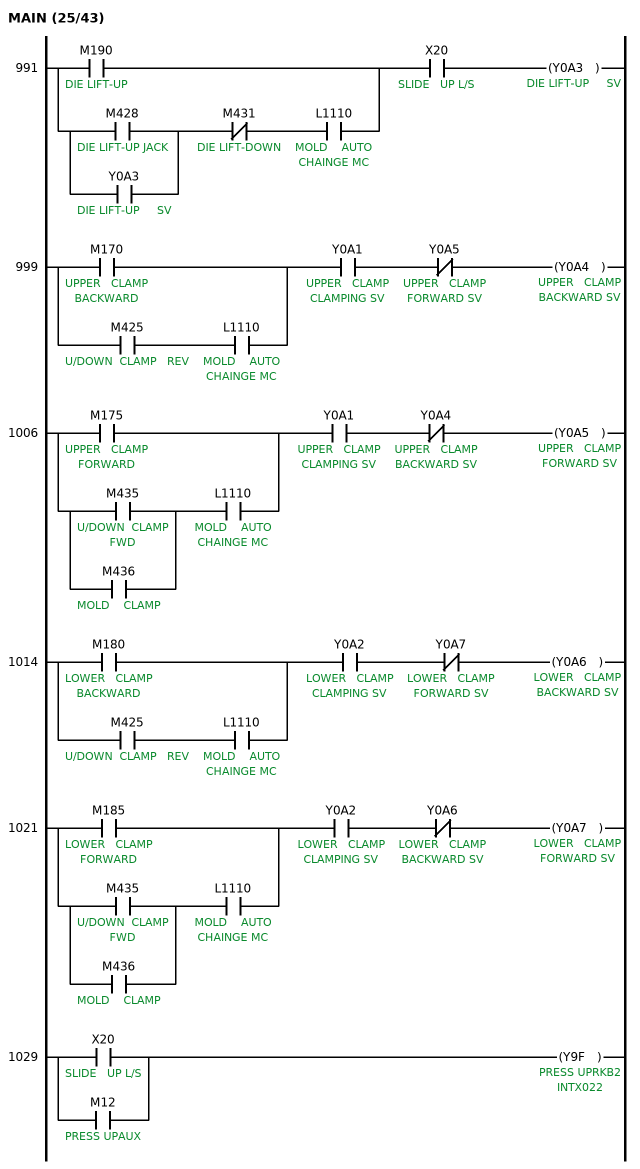
[picture p24: ladder of MAIN, rungs at steps 991 to 1029]
991   LD      M190  ; DIE LIFT-UP
      LD      M428  ; DIE LIFT-UP JACK
      OR      Y0A3  ; DIE LIFT-UP     SV
      ANI     M431  ; DIE LIFT-DOWN
      AND     L1110  ; MOLD    AUTO    CHAINGE MC
      ORB
      AND     X20  ; SLIDE   UP L/S
      OUT     Y0A3  ; DIE LIFT-UP     SV
999   LD      M170  ; UPPER   CLAMP   BACKWARD
      LD      M425  ; U/DOWN  CLAMP   REV
      AND     L1110  ; MOLD    AUTO    CHAINGE MC
      ORB
      AND     Y0A1  ; UPPER   CLAMP   CLAMPING SV
      ANI     Y0A5  ; UPPER   CLAMP   FORWARD SV
      OUT     Y0A4  ; UPPER   CLAMP   BACKWARD SV
1006  LD      M175  ; UPPER   CLAMP   FORWARD
      LD      M435  ; U/DOWN  CLAMP   FWD
      OR      M436  ; MOLD    CLAMP
      AND     L1110  ; MOLD    AUTO    CHAINGE MC
      ORB
      AND     Y0A1  ; UPPER   CLAMP   CLAMPING SV
      ANI     Y0A4  ; UPPER   CLAMP   BACKWARD SV
      OUT     Y0A5  ; UPPER   CLAMP   FORWARD SV
1014  LD      M180  ; LOWER   CLAMP   BACKWARD
      LD      M425  ; U/DOWN  CLAMP   REV
      AND     L1110  ; MOLD    AUTO    CHAINGE MC
      ORB
      AND     Y0A2  ; LOWER   CLAMP   CLAMPING SV
      ANI     Y0A7  ; LOWER   CLAMP   FORWARD SV
      OUT     Y0A6  ; LOWER   CLAMP   BACKWARD SV
1021  LD      M185  ; LOWER   CLAMP   FORWARD
      LD      M435  ; U/DOWN  CLAMP   FWD
      OR      M436  ; MOLD    CLAMP
      AND     L1110  ; MOLD    AUTO    CHAINGE MC
      ORB
      AND     Y0A2  ; LOWER   CLAMP   CLAMPING SV
      ANI     Y0A6  ; LOWER   CLAMP   BACKWARD SV
      OUT     Y0A7  ; LOWER   CLAMP   FORWARD SV
1029  LD      X20  ; SLIDE   UP L/S
      OR      M12  ; PRESS UPAUX
      OUT     Y9F  ; PRESS UPRKB2 INTX022
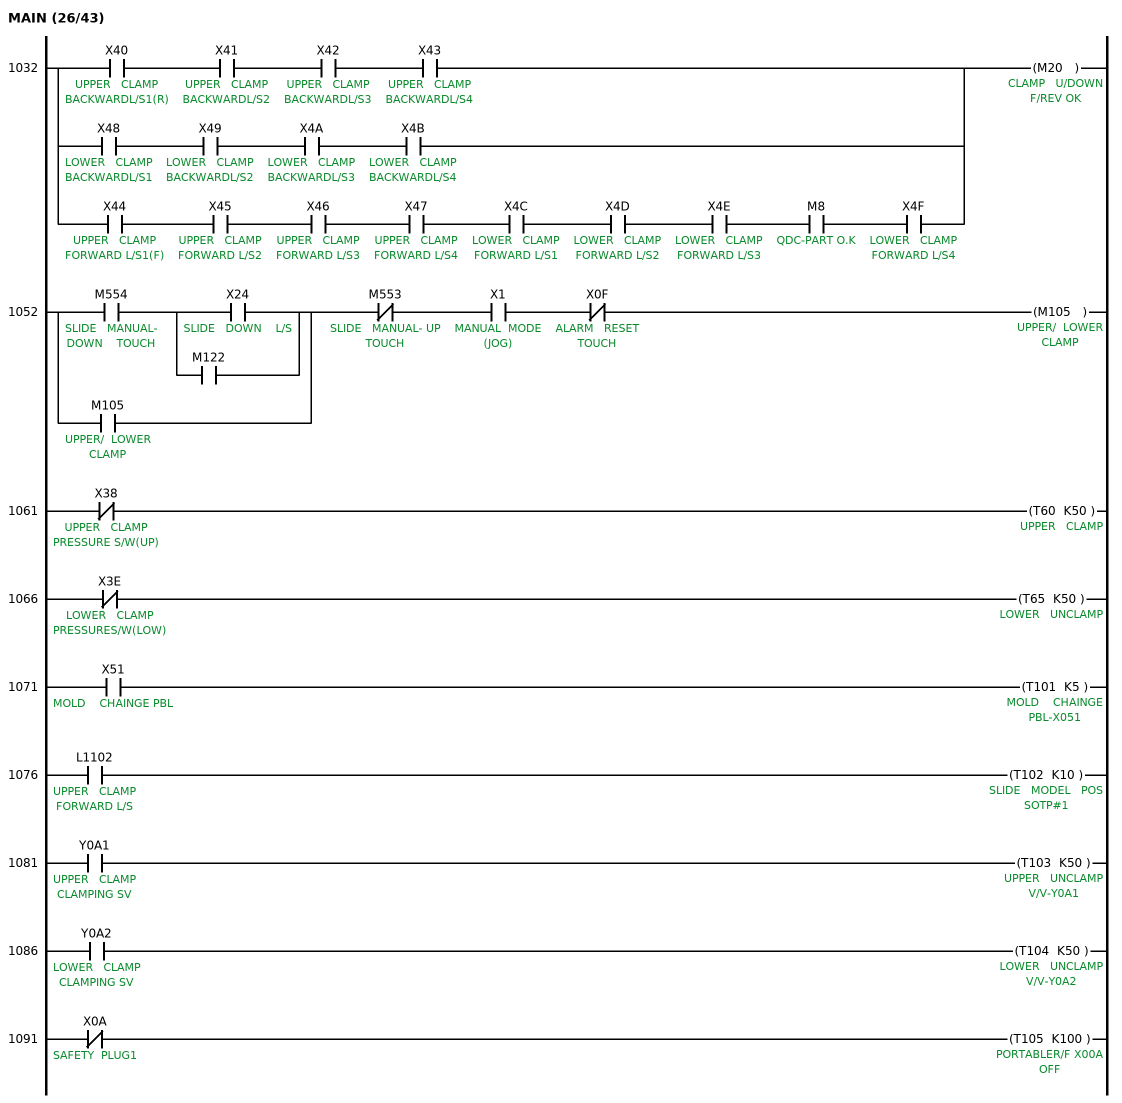
1032  LD      X40  ; UPPER   CLAMP   BACKWARDL/S1(R)
      AND     X41  ; UPPER   CLAMP   BACKWARDL/S2
      AND     X42  ; UPPER   CLAMP   BACKWARDL/S3
      AND     X43  ; UPPER   CLAMP   BACKWARDL/S4
      LD      X48  ; LOWER   CLAMP   BACKWARDL/S1
      AND     X49  ; LOWER   CLAMP   BACKWARDL/S2
      AND     X4A  ; LOWER   CLAMP   BACKWARDL/S3
      AND     X4B  ; LOWER   CLAMP   BACKWARDL/S4
      ORB
      LD      X44  ; UPPER   CLAMP   FORWARD L/S1(F)
      AND     X45  ; UPPER   CLAMP   FORWARD L/S2
      AND     X46  ; UPPER   CLAMP   FORWARD L/S3
      AND     X47  ; UPPER   CLAMP   FORWARD L/S4
      AND     X4C  ; LOWER   CLAMP   FORWARD L/S1
      AND     X4D  ; LOWER   CLAMP   FORWARD L/S2
      AND     X4E  ; LOWER   CLAMP   FORWARD L/S3
      AND     M8  ; QDC-PART O.K
      AND     X4F  ; LOWER   CLAMP   FORWARD L/S4
      ORB
      OUT     M20  ; CLAMP   U/DOWN  F/REV OK
1052  LD      M554  ; SLIDE   MANUAL- DOWN    TOUCH
      LD      X24  ; SLIDE   DOWN    L/S
      OR      M122
      ANB
      OR      M105  ; UPPER/  LOWER   CLAMP
      ANI     M553  ; SLIDE   MANUAL- UP      TOUCH
      AND     X1  ; MANUAL  MODE    (JOG)
      ANI     X0F  ; ALARM   RESET   TOUCH
      OUT     M105  ; UPPER/  LOWER   CLAMP
1061  LDI     X38  ; UPPER   CLAMP   PRESSURE S/W(UP)
      OUT     T60 K50  ; UPPER   CLAMP
1066  LDI     X3E  ; LOWER   CLAMP   PRESSURES/W(LOW)
      OUT     T65 K50  ; LOWER   UNCLAMP
1071  LD      X51  ; MOLD    CHAINGE PBL
      OUT     T101 K5  ; MOLD    CHAINGE PBL-X051
1076  LD      L1102  ; UPPER   CLAMP   FORWARD L/S
      OUT     T102 K10  ; SLIDE   MODEL   POS SOTP#1
1081  LD      Y0A1  ; UPPER   CLAMP   CLAMPING SV
      OUT     T103 K50  ; UPPER   UNCLAMP V/V-Y0A1
1086  LD      Y0A2  ; LOWER   CLAMP   CLAMPING SV
      OUT     T104 K50  ; LOWER   UNCLAMP V/V-Y0A2
1091  LDI     X0A  ; SAFETY  PLUG1
      OUT     T105 K100  ; PORTABLER/F X00A OFF
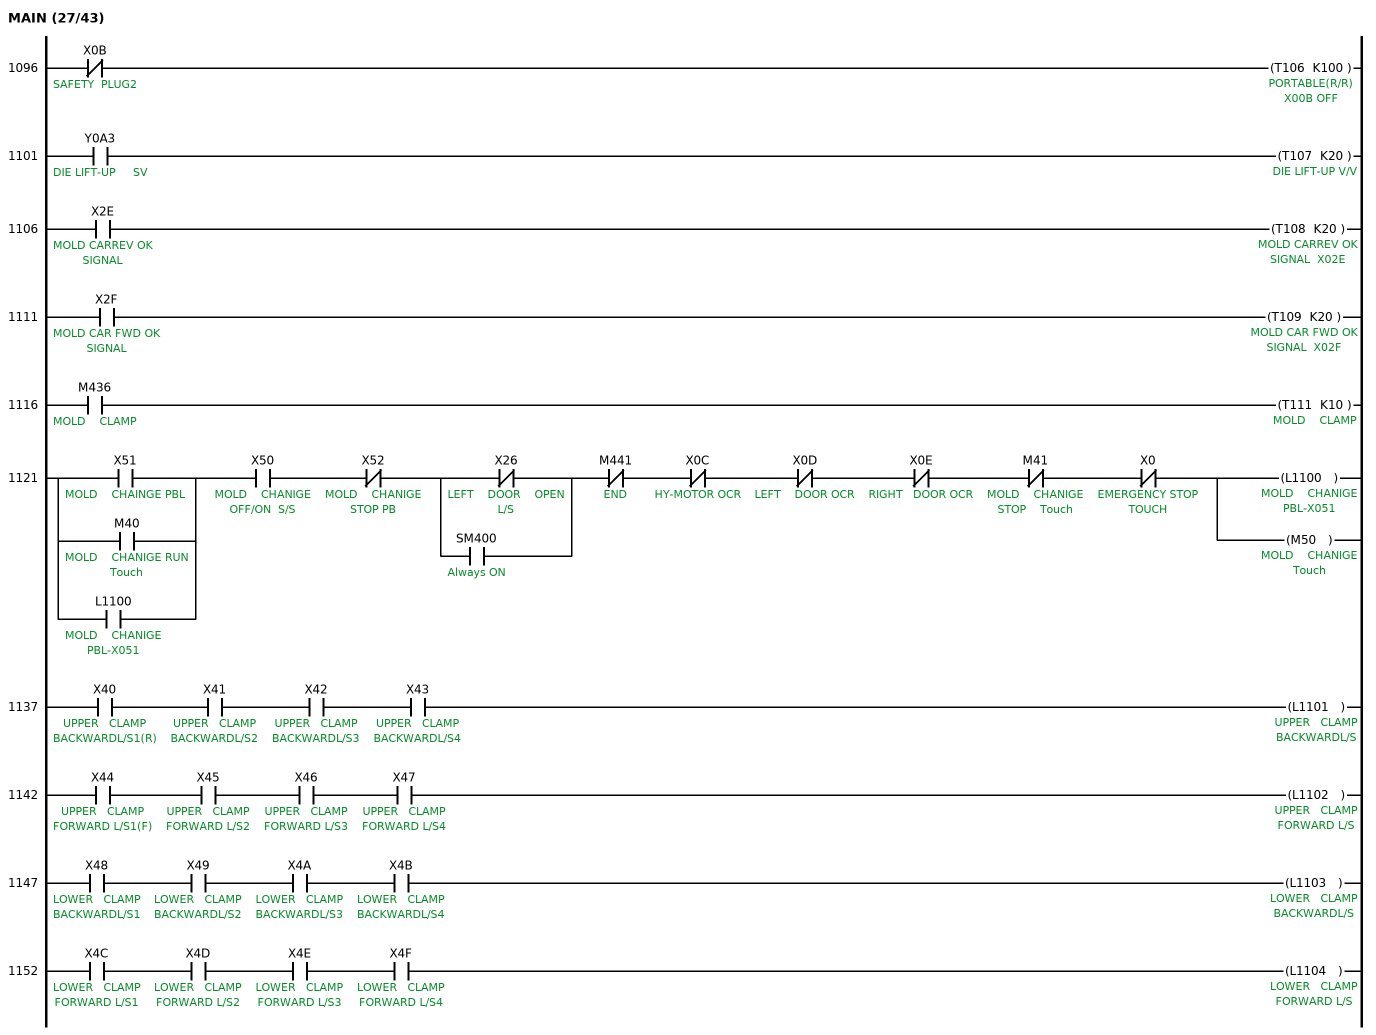
1096  LDI     X0B  ; SAFETY  PLUG2
      OUT     T106 K100  ; PORTABLE(R/R)   X00B OFF
1101  LD      Y0A3  ; DIE LIFT-UP     SV
      OUT     T107 K20  ; DIE LIFT-UP V/V
1106  LD      X2E  ; MOLD CARREV OK  SIGNAL
      OUT     T108 K20  ; MOLD CARREV OK  SIGNAL  X02E
1111  LD      X2F  ; MOLD CAR FWD OK  SIGNAL
      OUT     T109 K20  ; MOLD CAR FWD OK  SIGNAL  X02F
1116  LD      M436  ; MOLD    CLAMP
      OUT     T111 K10  ; MOLD    CLAMP
1121  LD      X51  ; MOLD    CHAINGE PBL
      OR      M40  ; MOLD    CHANIGE RUN     Touch
      OR      L1100  ; MOLD    CHANIGE PBL-X051
      AND     X50  ; MOLD    CHANIGE OFF/ON  S/S
      ANI     X52  ; MOLD    CHANIGE STOP PB
      LDI     X26  ; LEFT    DOOR    OPEN L/S
      OR      SM400  ; Always ON
      ANB
      ANI     M441  ; END
      ANI     X0C  ; HY-MOTOR OCR
      ANI     X0D  ; LEFT    DOOR OCR
      ANI     X0E  ; RIGHT   DOOR OCR
      ANI     M41  ; MOLD    CHANIGE STOP    Touch
      ANI     X0  ; EMERGENCY STOP  TOUCH
      OUT     L1100  ; MOLD    CHANIGE PBL-X051
      OUT     M50  ; MOLD    CHANIGE Touch
1137  LD      X40  ; UPPER   CLAMP   BACKWARDL/S1(R)
      AND     X41  ; UPPER   CLAMP   BACKWARDL/S2
      AND     X42  ; UPPER   CLAMP   BACKWARDL/S3
      AND     X43  ; UPPER   CLAMP   BACKWARDL/S4
      OUT     L1101  ; UPPER   CLAMP   BACKWARDL/S
1142  LD      X44  ; UPPER   CLAMP   FORWARD L/S1(F)
      AND     X45  ; UPPER   CLAMP   FORWARD L/S2
      AND     X46  ; UPPER   CLAMP   FORWARD L/S3
      AND     X47  ; UPPER   CLAMP   FORWARD L/S4
      OUT     L1102  ; UPPER   CLAMP   FORWARD L/S
1147  LD      X48  ; LOWER   CLAMP   BACKWARDL/S1
      AND     X49  ; LOWER   CLAMP   BACKWARDL/S2
      AND     X4A  ; LOWER   CLAMP   BACKWARDL/S3
      AND     X4B  ; LOWER   CLAMP   BACKWARDL/S4
      OUT     L1103  ; LOWER   CLAMP   BACKWARDL/S
1152  LD      X4C  ; LOWER   CLAMP   FORWARD L/S1
      AND     X4D  ; LOWER   CLAMP   FORWARD L/S2
      AND     X4E  ; LOWER   CLAMP   FORWARD L/S3
      AND     X4F  ; LOWER   CLAMP   FORWARD L/S4
      OUT     L1104  ; LOWER   CLAMP   FORWARD L/S
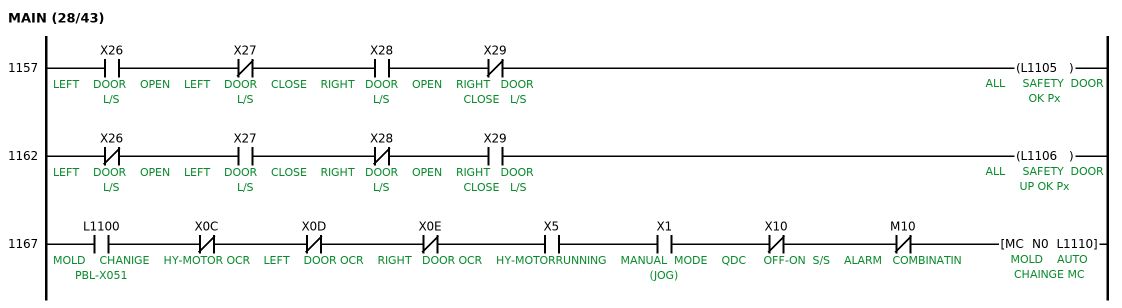
1157  LD      X26  ; LEFT    DOOR    OPEN L/S
      ANI     X27  ; LEFT    DOOR    CLOSE   L/S
      AND     X28  ; RIGHT   DOOR    OPEN L/S
      ANI     X29  ; RIGHT   DOOR    CLOSE   L/S
      OUT     L1105  ; ALL     SAFETY  DOOR OK Px
1162  LDI     X26  ; LEFT    DOOR    OPEN L/S
      AND     X27  ; LEFT    DOOR    CLOSE   L/S
      ANI     X28  ; RIGHT   DOOR    OPEN L/S
      AND     X29  ; RIGHT   DOOR    CLOSE   L/S
      OUT     L1106  ; ALL     SAFETY  DOOR UP OK Px
1167  LD      L1100  ; MOLD    CHANIGE PBL-X051
      ANI     X0C  ; HY-MOTOR OCR
      ANI     X0D  ; LEFT    DOOR OCR
      ANI     X0E  ; RIGHT   DOOR OCR
      AND     X5  ; HY-MOTORRUNNING
      AND     X1  ; MANUAL  MODE    (JOG)
      ANI     X10  ; QDC     OFF-ON  S/S
      ANI     M10  ; ALARM   COMBINATIN
      MC      N0 L1110
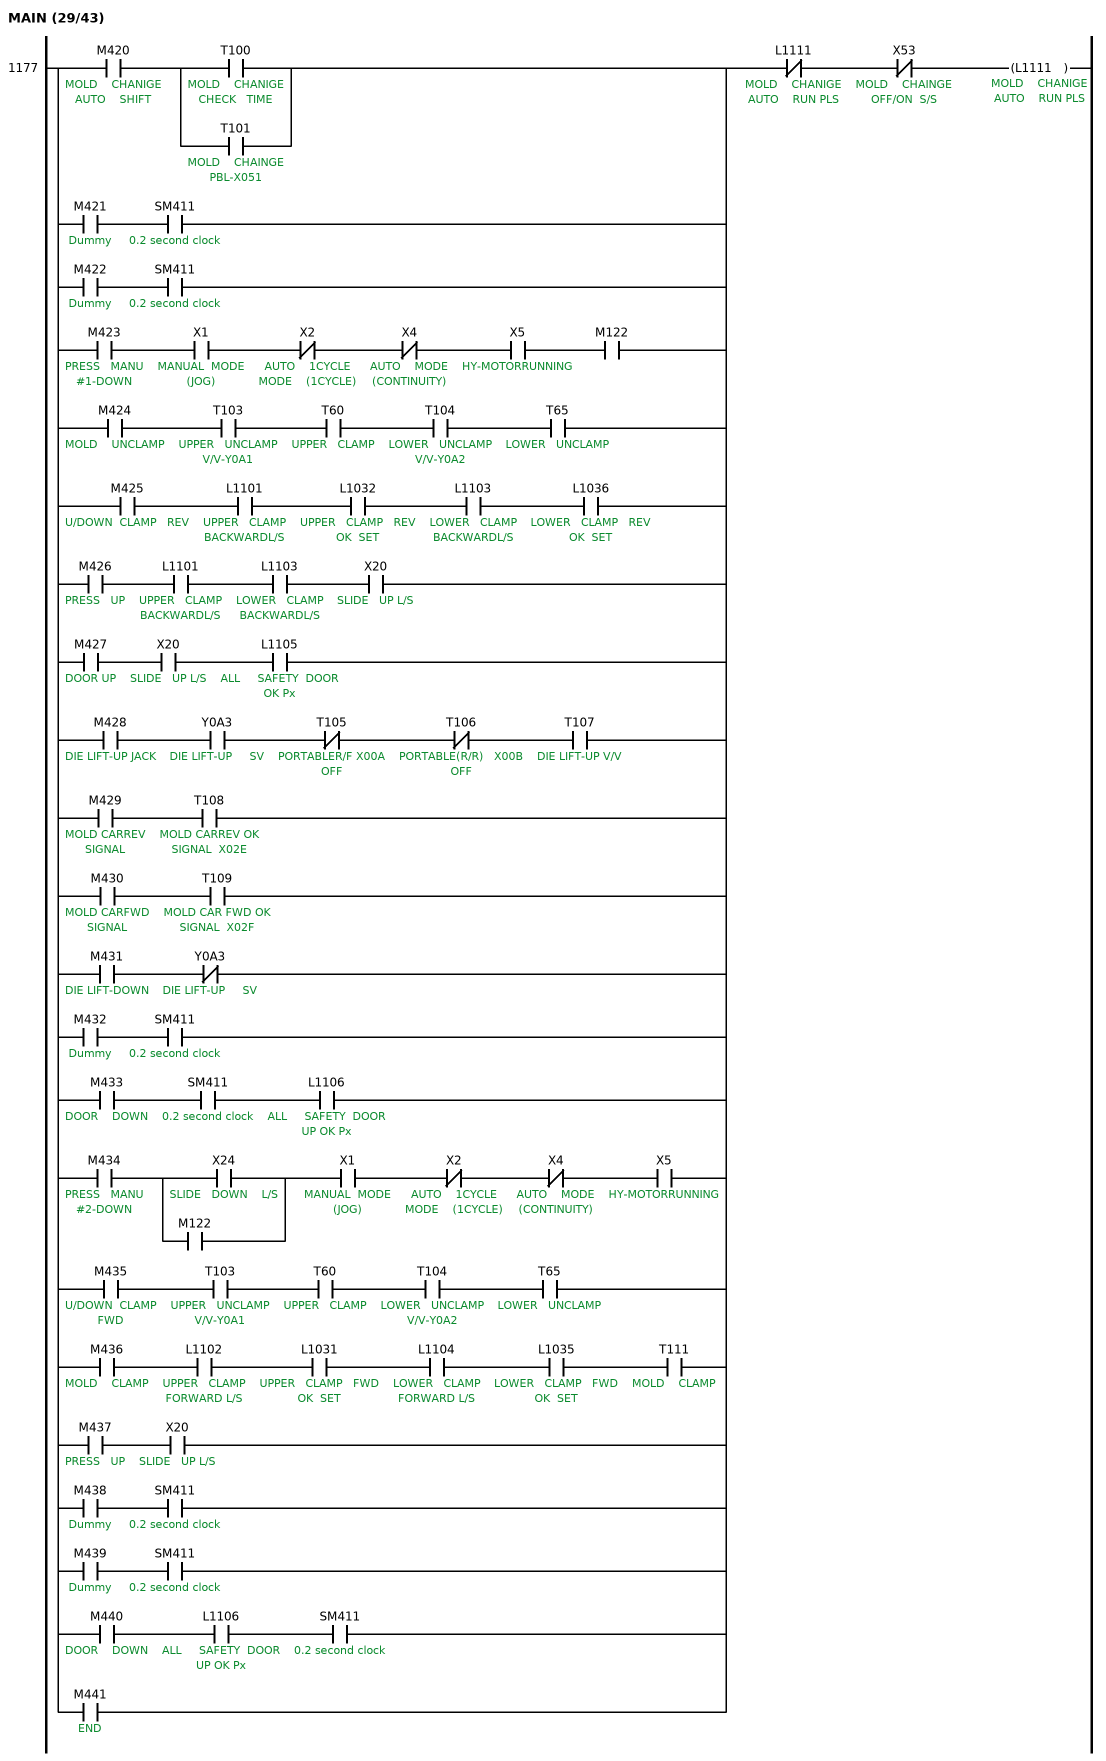
1177  LD      M420  ; MOLD    CHANIGE AUTO    SHIFT
      LD      T100  ; MOLD    CHANIGE CHECK   TIME
      OR      T101  ; MOLD    CHAINGE PBL-X051
      ANB
      LD      M421  ; Dummy
      AND     SM411  ; 0.2 second clock
      ORB
      LD      M422  ; Dummy
      AND     SM411  ; 0.2 second clock
      ORB
      LD      M423  ; PRESS   MANU #1-DOWN
      AND     X1  ; MANUAL  MODE    (JOG)
      ANI     X2  ; AUTO    1CYCLE  MODE    (1CYCLE)
      ANI     X4  ; AUTO    MODE    (CONTINUITY)
      AND     X5  ; HY-MOTORRUNNING
      AND     M122
      ORB
      LD      M424  ; MOLD    UNCLAMP
      AND     T103  ; UPPER   UNCLAMP V/V-Y0A1
      AND     T60  ; UPPER   CLAMP
      AND     T104  ; LOWER   UNCLAMP V/V-Y0A2
      AND     T65  ; LOWER   UNCLAMP
      ORB
      LD      M425  ; U/DOWN  CLAMP   REV
      AND     L1101  ; UPPER   CLAMP   BACKWARDL/S
      AND     L1032  ; UPPER   CLAMP   REV OK  SET
      AND     L1103  ; LOWER   CLAMP   BACKWARDL/S
      AND     L1036  ; LOWER   CLAMP   REV OK  SET
      ORB
      LD      M426  ; PRESS   UP
      AND     L1101  ; UPPER   CLAMP   BACKWARDL/S
      AND     L1103  ; LOWER   CLAMP   BACKWARDL/S
      AND     X20  ; SLIDE   UP L/S
      ORB
      LD      M427  ; DOOR UP
      AND     X20  ; SLIDE   UP L/S
      AND     L1105  ; ALL     SAFETY  DOOR OK Px
      ORB
      LD      M428  ; DIE LIFT-UP JACK
      AND     Y0A3  ; DIE LIFT-UP     SV
      ANI     T105  ; PORTABLER/F X00A OFF
      ANI     T106  ; PORTABLE(R/R)   X00B OFF
      AND     T107  ; DIE LIFT-UP V/V
      ORB
      LD      M429  ; MOLD CARREV     SIGNAL
      AND     T108  ; MOLD CARREV OK  SIGNAL  X02E
      ORB
      LD      M430  ; MOLD CARFWD     SIGNAL
      AND     T109  ; MOLD CAR FWD OK  SIGNAL  X02F
      ORB
      LD      M431  ; DIE LIFT-DOWN
      ANI     Y0A3  ; DIE LIFT-UP     SV
      ORB
      LD      M432  ; Dummy
      AND     SM411  ; 0.2 second clock
      ORB
      LD      M433  ; DOOR    DOWN
      AND     SM411  ; 0.2 second clock
      AND     L1106  ; ALL     SAFETY  DOOR UP OK Px
      ORB
      LD      M434  ; PRESS   MANU #2-DOWN
      LD      X24  ; SLIDE   DOWN    L/S
      OR      M122
      ANB
      AND     X1  ; MANUAL  MODE    (JOG)
      ANI     X2  ; AUTO    1CYCLE  MODE    (1CYCLE)
      ANI     X4  ; AUTO    MODE    (CONTINUITY)
      AND     X5  ; HY-MOTORRUNNING
      ORB
      LD      M435  ; U/DOWN  CLAMP   FWD
      AND     T103  ; UPPER   UNCLAMP V/V-Y0A1
      AND     T60  ; UPPER   CLAMP
      AND     T104  ; LOWER   UNCLAMP V/V-Y0A2
      AND     T65  ; LOWER   UNCLAMP
      ORB
      LD      M436  ; MOLD    CLAMP
      AND     L1102  ; UPPER   CLAMP   FORWARD L/S
      AND     L1031  ; UPPER   CLAMP   FWD OK  SET
      AND     L1104  ; LOWER   CLAMP   FORWARD L/S
      AND     L1035  ; LOWER   CLAMP   FWD OK  SET
      AND     T111  ; MOLD    CLAMP
      ORB
      LD      M437  ; PRESS   UP
      AND     X20  ; SLIDE   UP L/S
      ORB
      LD      M438  ; Dummy
      AND     SM411  ; 0.2 second clock
      ORB
      LD      M439  ; Dummy
      AND     SM411  ; 0.2 second clock
      ORB
      LD      M440  ; DOOR    DOWN
      AND     L1106  ; ALL     SAFETY  DOOR UP OK Px
      AND     SM411  ; 0.2 second clock
      ORB
      OR      M441  ; END
      ANI     L1111  ; MOLD    CHANIGE AUTO    RUN PLS
      ANI     X53  ; MOLD    CHAINGE OFF/ON  S/S
      OUT     L1111  ; MOLD    CHANIGE AUTO    RUN PLS
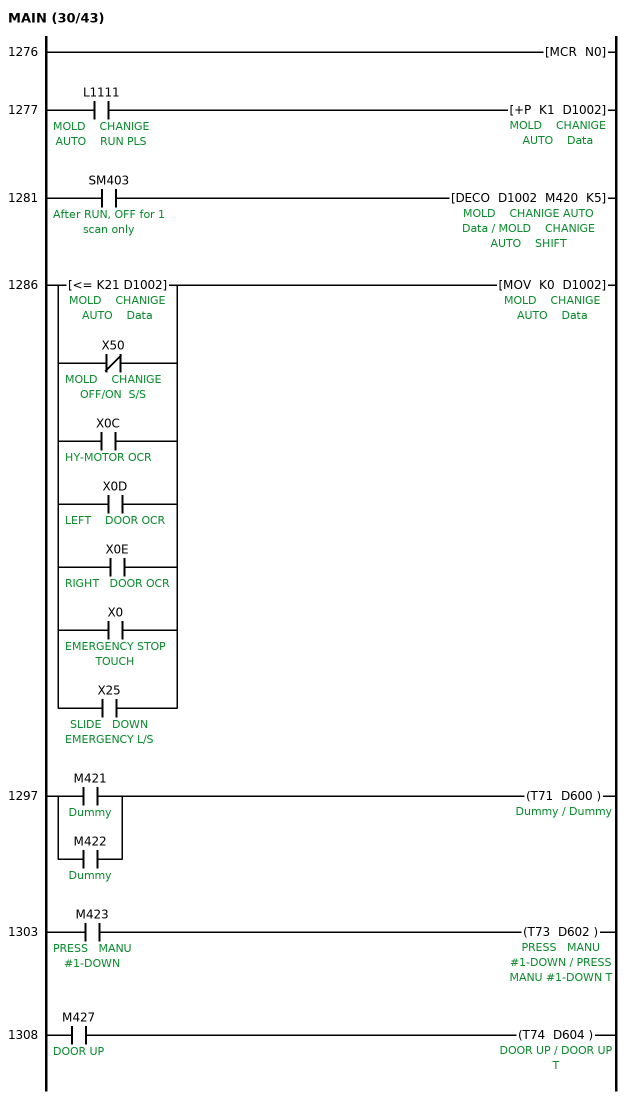
1276  MCR     N0
1277  LD      L1111  ; MOLD    CHANIGE AUTO    RUN PLS
      +P      K1 D1002
1281  LD      SM403  ; After RUN, OFF for 1 scan only
      DECO    D1002 M420 K5
1286  LD<=    K21 D1002  ; MOLD    CHANIGE AUTO    Data
      ORI     X50  ; MOLD    CHANIGE OFF/ON  S/S
      OR      X0C  ; HY-MOTOR OCR
      OR      X0D  ; LEFT    DOOR OCR
      OR      X0E  ; RIGHT   DOOR OCR
      OR      X0  ; EMERGENCY STOP  TOUCH
      OR      X25  ; SLIDE   DOWN    EMERGENCY L/S
      MOV     K0 D1002
1297  LD      M421  ; Dummy
      OR      M422  ; Dummy
      OUT     T71 D600  ; Dummy / Dummy
1303  LD      M423  ; PRESS   MANU #1-DOWN
      OUT     T73 D602  ; PRESS   MANU #1-DOWN / PRESS   MANU #1-DOWN T
1308  LD      M427  ; DOOR UP
      OUT     T74 D604  ; DOOR UP / DOOR UP T
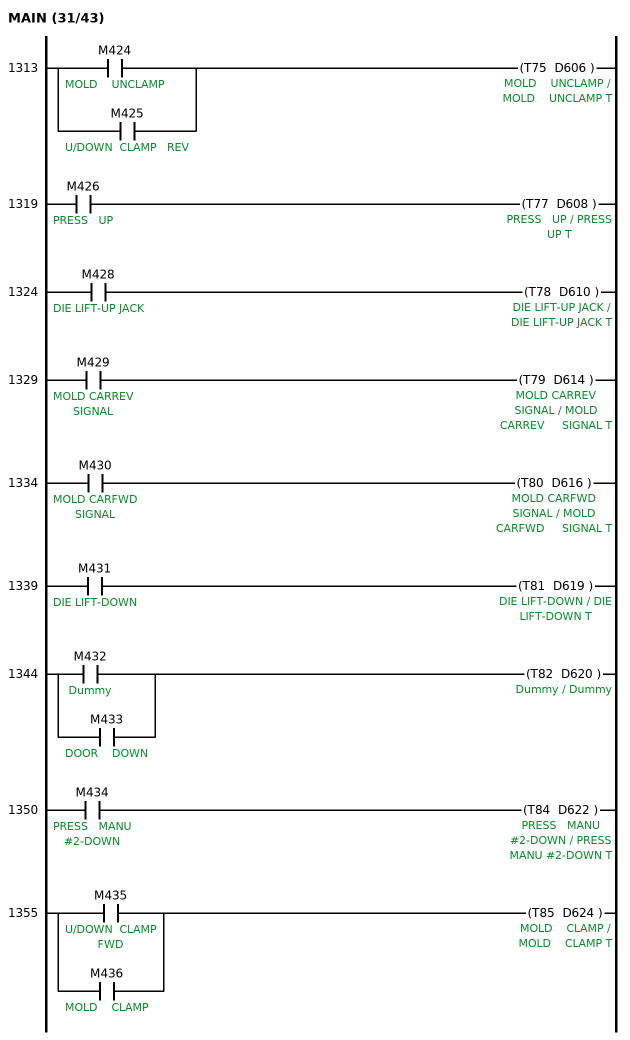
1313  LD      M424  ; MOLD    UNCLAMP
      OR      M425  ; U/DOWN  CLAMP   REV
      OUT     T75 D606  ; MOLD    UNCLAMP / MOLD    UNCLAMP T
1319  LD      M426  ; PRESS   UP
      OUT     T77 D608  ; PRESS   UP / PRESS   UP T
1324  LD      M428  ; DIE LIFT-UP JACK
      OUT     T78 D610  ; DIE LIFT-UP JACK / DIE LIFT-UP JACK T
1329  LD      M429  ; MOLD CARREV     SIGNAL
      OUT     T79 D614  ; MOLD CARREV     SIGNAL / MOLD CARREV     SIGNAL T
1334  LD      M430  ; MOLD CARFWD     SIGNAL
      OUT     T80 D616  ; MOLD CARFWD     SIGNAL / MOLD CARFWD     SIGNAL T
1339  LD      M431  ; DIE LIFT-DOWN
      OUT     T81 D619  ; DIE LIFT-DOWN / DIE LIFT-DOWN T
1344  LD      M432  ; Dummy
      OR      M433  ; DOOR    DOWN
      OUT     T82 D620  ; Dummy / Dummy
1350  LD      M434  ; PRESS   MANU #2-DOWN
      OUT     T84 D622  ; PRESS   MANU #2-DOWN / PRESS   MANU #2-DOWN T
1355  LD      M435  ; U/DOWN  CLAMP   FWD
      OR      M436  ; MOLD    CLAMP
      OUT     T85 D624  ; MOLD    CLAMP / MOLD    CLAMP T
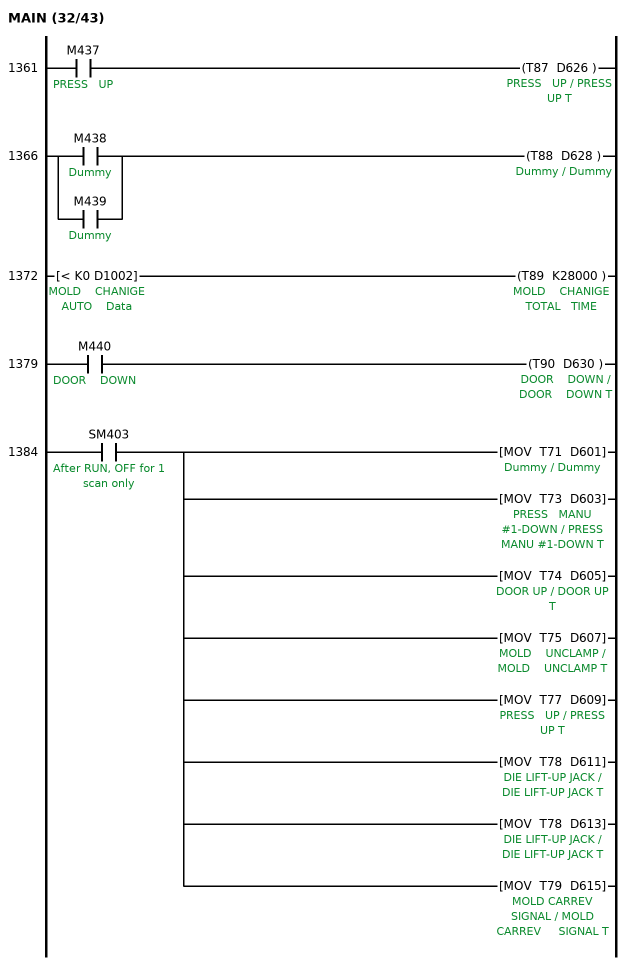
1361  LD      M437  ; PRESS   UP
      OUT     T87 D626  ; PRESS   UP / PRESS   UP T
1366  LD      M438  ; Dummy
      OR      M439  ; Dummy
      OUT     T88 D628  ; Dummy / Dummy
1372  LD<     K0 D1002  ; MOLD    CHANIGE AUTO    Data
      OUT     T89 K28000  ; MOLD    CHANIGE TOTAL   TIME
1379  LD      M440  ; DOOR    DOWN
      OUT     T90 D630  ; DOOR    DOWN / DOOR    DOWN T
1384  LD      SM403  ; After RUN, OFF for 1 scan only
      MOV     T71 D601  ; Dummy
      MOV     T73 D603  ; PRESS   MANU #1-DOWN T
      MOV     T74 D605  ; DOOR UP T
      MOV     T75 D607  ; MOLD    UNCLAMP T
      MOV     T77 D609  ; PRESS   UP T
      MOV     T78 D611  ; DIE LIFT-UP JACK T
      MOV     T78 D613  ; DIE LIFT-UP JACK T
      MOV     T79 D615  ; MOLD CARREV     SIGNAL T
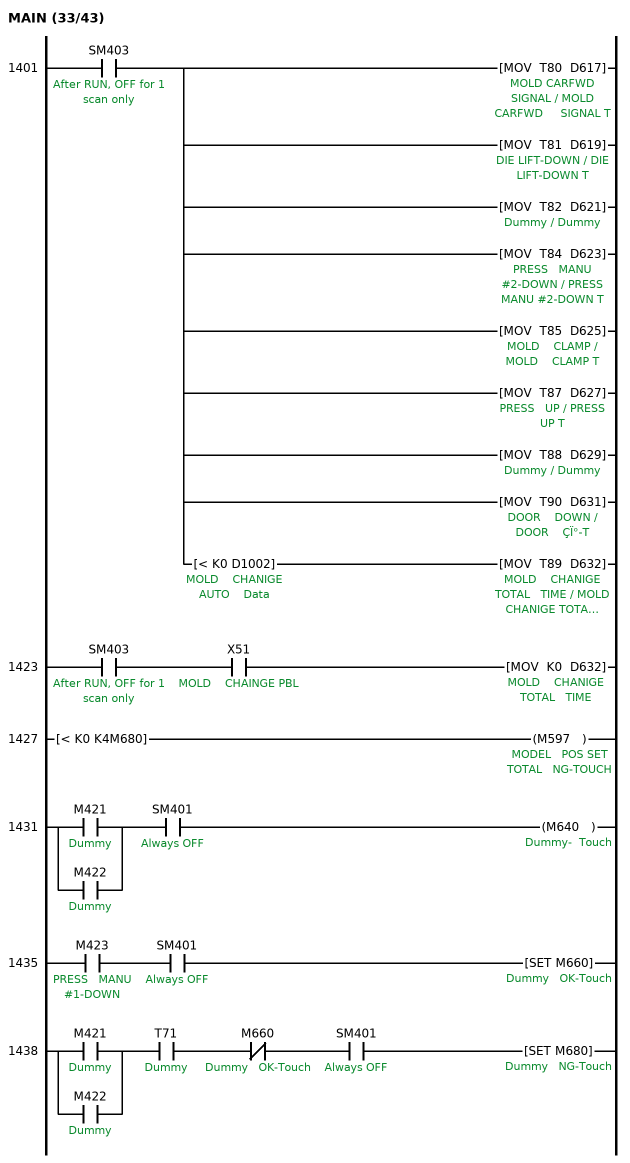
1401  LD      SM403  ; After RUN, OFF for 1 scan only
      MOV     T80 D617  ; MOLD CARFWD     SIGNAL T
      MOV     T81 D619
      MOV     T82 D621  ; Dummy
      MOV     T84 D623  ; PRESS   MANU #2-DOWN T
      MOV     T85 D625  ; MOLD    CLAMP T
      MOV     T87 D627  ; PRESS   UP T
      MOV     T88 D629  ; Dummy
      MOV     T90 D631  ; DOOR    ÇÏ°­T
      AND<    K0 D1002  ; MOLD    CHANIGE AUTO    Data
      MOV     T89 D632  ; MOLD    CHANIGE TOTAL   TIME
1423  LD      SM403  ; After RUN, OFF for 1 scan only
      AND     X51  ; MOLD    CHAINGE PBL
      MOV     K0 D632
1427  LD<     K0 K4M680  ; Dummy   NG-Touch
      OUT     M597  ; MODEL   POS SET TOTAL   NG-TOUCH
1431  LD      M421  ; Dummy
      OR      M422  ; Dummy
      AND     SM401  ; Always OFF
      OUT     M640  ; Dummy-  Touch
1435  LD      M423  ; PRESS   MANU #1-DOWN
      AND     SM401  ; Always OFF
      SET     M660  ; Dummy   OK-Touch
1438  LD      M421  ; Dummy
      OR      M422  ; Dummy
      AND     T71  ; Dummy
      ANI     M660  ; Dummy   OK-Touch
      AND     SM401  ; Always OFF
      SET     M680  ; Dummy   NG-Touch
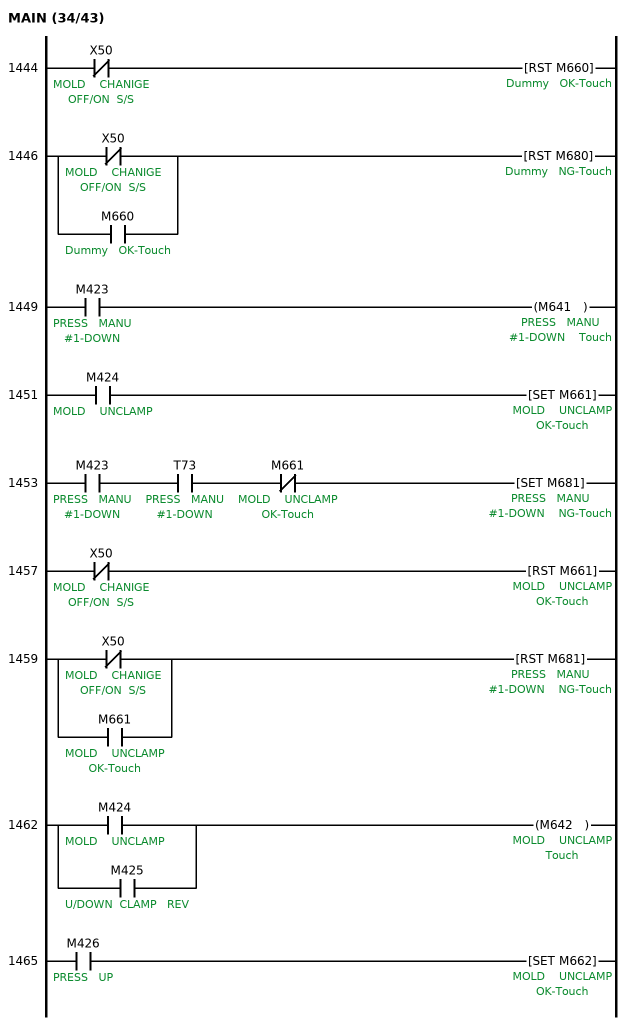
1444  LDI     X50  ; MOLD    CHANIGE OFF/ON  S/S
      RST     M660  ; Dummy   OK-Touch
1446  LDI     X50  ; MOLD    CHANIGE OFF/ON  S/S
      OR      M660  ; Dummy   OK-Touch
      RST     M680  ; Dummy   NG-Touch
1449  LD      M423  ; PRESS   MANU #1-DOWN
      OUT     M641  ; PRESS   MANU #1-DOWN    Touch
1451  LD      M424  ; MOLD    UNCLAMP
      SET     M661  ; MOLD    UNCLAMP OK-Touch
1453  LD      M423  ; PRESS   MANU #1-DOWN
      AND     T73  ; PRESS   MANU #1-DOWN
      ANI     M661  ; MOLD    UNCLAMP OK-Touch
      SET     M681  ; PRESS   MANU #1-DOWN    NG-Touch
1457  LDI     X50  ; MOLD    CHANIGE OFF/ON  S/S
      RST     M661  ; MOLD    UNCLAMP OK-Touch
1459  LDI     X50  ; MOLD    CHANIGE OFF/ON  S/S
      OR      M661  ; MOLD    UNCLAMP OK-Touch
      RST     M681  ; PRESS   MANU #1-DOWN    NG-Touch
1462  LD      M424  ; MOLD    UNCLAMP
      OR      M425  ; U/DOWN  CLAMP   REV
      OUT     M642  ; MOLD    UNCLAMP Touch
1465  LD      M426  ; PRESS   UP
      SET     M662  ; MOLD    UNCLAMP OK-Touch
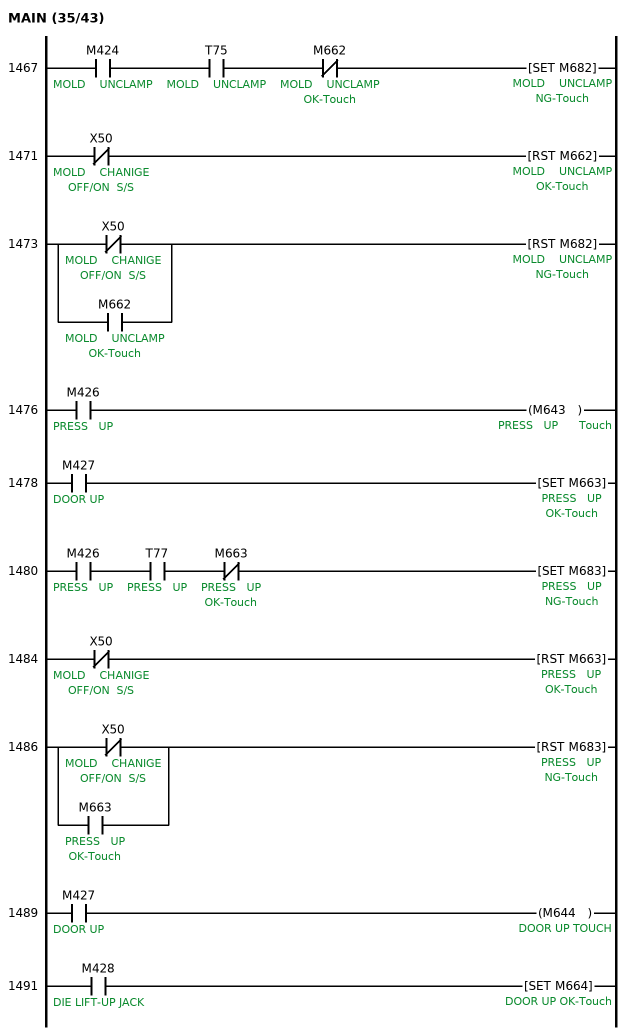
1467  LD      M424  ; MOLD    UNCLAMP
      AND     T75  ; MOLD    UNCLAMP
      ANI     M662  ; MOLD    UNCLAMP OK-Touch
      SET     M682  ; MOLD    UNCLAMP NG-Touch
1471  LDI     X50  ; MOLD    CHANIGE OFF/ON  S/S
      RST     M662  ; MOLD    UNCLAMP OK-Touch
1473  LDI     X50  ; MOLD    CHANIGE OFF/ON  S/S
      OR      M662  ; MOLD    UNCLAMP OK-Touch
      RST     M682  ; MOLD    UNCLAMP NG-Touch
1476  LD      M426  ; PRESS   UP
      OUT     M643  ; PRESS   UP      Touch
1478  LD      M427  ; DOOR UP
      SET     M663  ; PRESS   UP      OK-Touch
1480  LD      M426  ; PRESS   UP
      AND     T77  ; PRESS   UP
      ANI     M663  ; PRESS   UP      OK-Touch
      SET     M683  ; PRESS   UP      NG-Touch
1484  LDI     X50  ; MOLD    CHANIGE OFF/ON  S/S
      RST     M663  ; PRESS   UP      OK-Touch
1486  LDI     X50  ; MOLD    CHANIGE OFF/ON  S/S
      OR      M663  ; PRESS   UP      OK-Touch
      RST     M683  ; PRESS   UP      NG-Touch
1489  LD      M427  ; DOOR UP
      OUT     M644  ; DOOR UP TOUCH
1491  LD      M428  ; DIE LIFT-UP JACK
      SET     M664  ; DOOR UP OK-Touch
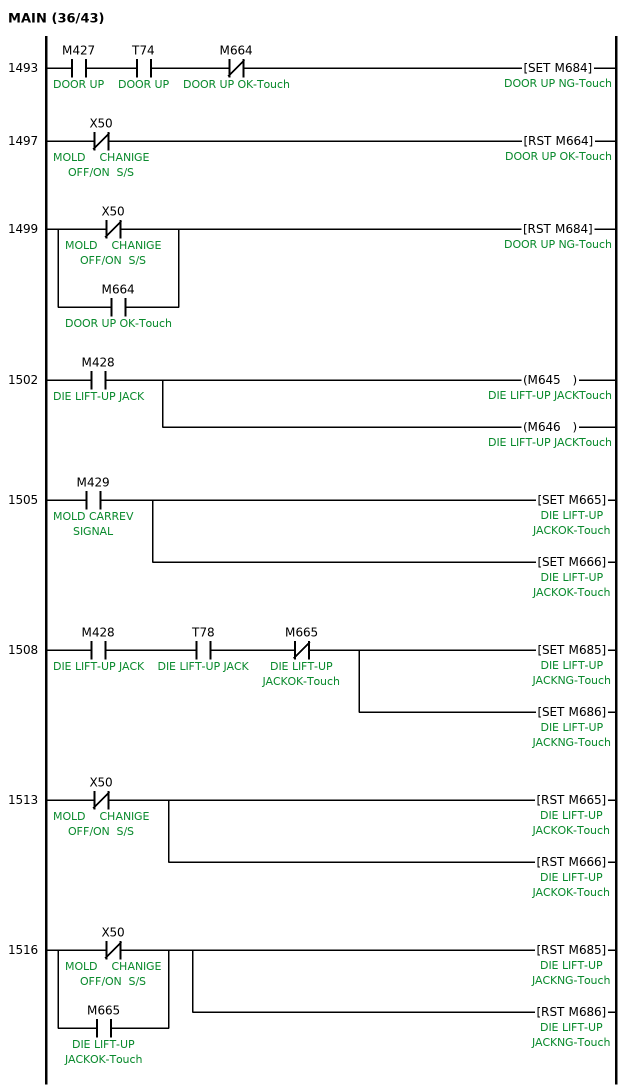
1493  LD      M427  ; DOOR UP
      AND     T74  ; DOOR UP
      ANI     M664  ; DOOR UP OK-Touch
      SET     M684  ; DOOR UP NG-Touch
1497  LDI     X50  ; MOLD    CHANIGE OFF/ON  S/S
      RST     M664  ; DOOR UP OK-Touch
1499  LDI     X50  ; MOLD    CHANIGE OFF/ON  S/S
      OR      M664  ; DOOR UP OK-Touch
      RST     M684  ; DOOR UP NG-Touch
1502  LD      M428  ; DIE LIFT-UP JACK
      OUT     M645  ; DIE LIFT-UP JACKTouch
      OUT     M646  ; DIE LIFT-UP JACKTouch
1505  LD      M429  ; MOLD CARREV     SIGNAL
      SET     M665  ; DIE LIFT-UP JACKOK-Touch
      SET     M666  ; DIE LIFT-UP JACKOK-Touch
1508  LD      M428  ; DIE LIFT-UP JACK
      AND     T78  ; DIE LIFT-UP JACK
      ANI     M665  ; DIE LIFT-UP JACKOK-Touch
      SET     M685  ; DIE LIFT-UP JACKNG-Touch
      SET     M686  ; DIE LIFT-UP JACKNG-Touch
1513  LDI     X50  ; MOLD    CHANIGE OFF/ON  S/S
      RST     M665  ; DIE LIFT-UP JACKOK-Touch
      RST     M666  ; DIE LIFT-UP JACKOK-Touch
1516  LDI     X50  ; MOLD    CHANIGE OFF/ON  S/S
      OR      M665  ; DIE LIFT-UP JACKOK-Touch
      RST     M685  ; DIE LIFT-UP JACKNG-Touch
      RST     M686  ; DIE LIFT-UP JACKNG-Touch
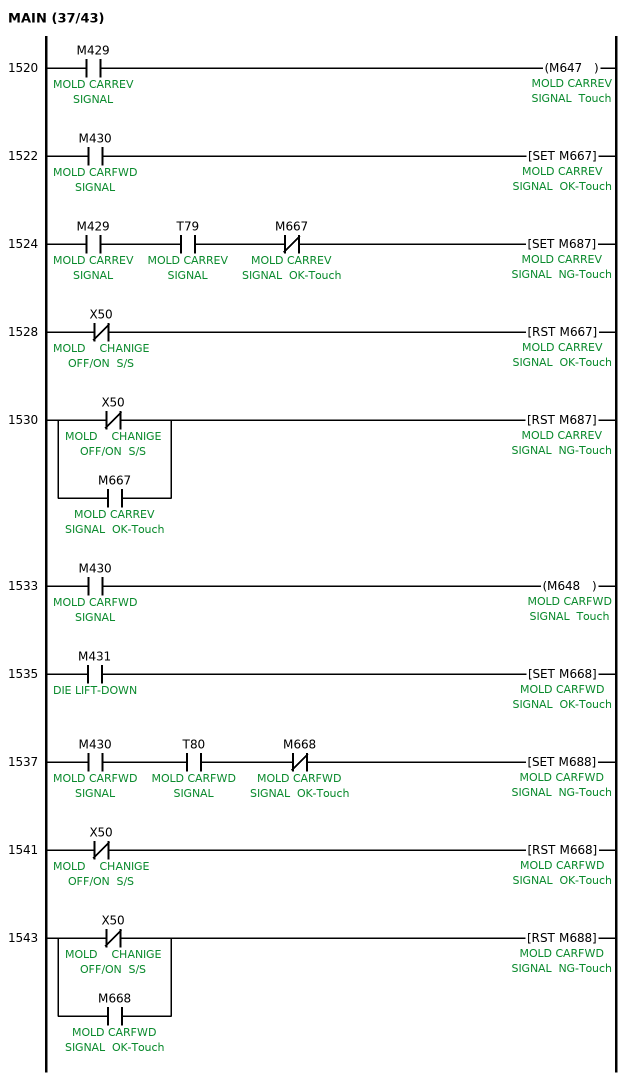
1520  LD      M429  ; MOLD CARREV     SIGNAL
      OUT     M647  ; MOLD CARREV     SIGNAL  Touch
1522  LD      M430  ; MOLD CARFWD     SIGNAL
      SET     M667  ; MOLD CARREV     SIGNAL  OK-Touch
1524  LD      M429  ; MOLD CARREV     SIGNAL
      AND     T79  ; MOLD CARREV     SIGNAL
      ANI     M667  ; MOLD CARREV     SIGNAL  OK-Touch
      SET     M687  ; MOLD CARREV     SIGNAL  NG-Touch
1528  LDI     X50  ; MOLD    CHANIGE OFF/ON  S/S
      RST     M667  ; MOLD CARREV     SIGNAL  OK-Touch
1530  LDI     X50  ; MOLD    CHANIGE OFF/ON  S/S
      OR      M667  ; MOLD CARREV     SIGNAL  OK-Touch
      RST     M687  ; MOLD CARREV     SIGNAL  NG-Touch
1533  LD      M430  ; MOLD CARFWD     SIGNAL
      OUT     M648  ; MOLD CARFWD     SIGNAL  Touch
1535  LD      M431  ; DIE LIFT-DOWN
      SET     M668  ; MOLD CARFWD     SIGNAL  OK-Touch
1537  LD      M430  ; MOLD CARFWD     SIGNAL
      AND     T80  ; MOLD CARFWD     SIGNAL
      ANI     M668  ; MOLD CARFWD     SIGNAL  OK-Touch
      SET     M688  ; MOLD CARFWD     SIGNAL  NG-Touch
1541  LDI     X50  ; MOLD    CHANIGE OFF/ON  S/S
      RST     M668  ; MOLD CARFWD     SIGNAL  OK-Touch
1543  LDI     X50  ; MOLD    CHANIGE OFF/ON  S/S
      OR      M668  ; MOLD CARFWD     SIGNAL  OK-Touch
      RST     M688  ; MOLD CARFWD     SIGNAL  NG-Touch
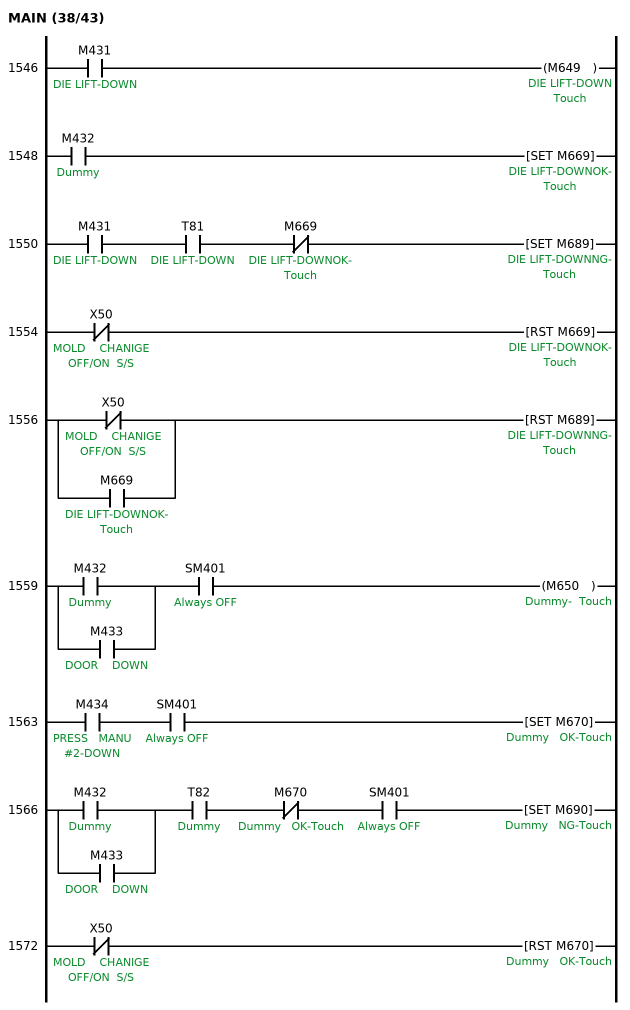
1546  LD      M431  ; DIE LIFT-DOWN
      OUT     M649  ; DIE LIFT-DOWN   Touch
1548  LD      M432  ; Dummy
      SET     M669  ; DIE LIFT-DOWNOK-Touch
1550  LD      M431  ; DIE LIFT-DOWN
      AND     T81  ; DIE LIFT-DOWN
      ANI     M669  ; DIE LIFT-DOWNOK-Touch
      SET     M689  ; DIE LIFT-DOWNNG-Touch
1554  LDI     X50  ; MOLD    CHANIGE OFF/ON  S/S
      RST     M669  ; DIE LIFT-DOWNOK-Touch
1556  LDI     X50  ; MOLD    CHANIGE OFF/ON  S/S
      OR      M669  ; DIE LIFT-DOWNOK-Touch
      RST     M689  ; DIE LIFT-DOWNNG-Touch
1559  LD      M432  ; Dummy
      OR      M433  ; DOOR    DOWN
      AND     SM401  ; Always OFF
      OUT     M650  ; Dummy-  Touch
1563  LD      M434  ; PRESS   MANU #2-DOWN
      AND     SM401  ; Always OFF
      SET     M670  ; Dummy   OK-Touch
1566  LD      M432  ; Dummy
      OR      M433  ; DOOR    DOWN
      AND     T82  ; Dummy
      ANI     M670  ; Dummy   OK-Touch
      AND     SM401  ; Always OFF
      SET     M690  ; Dummy   NG-Touch
1572  LDI     X50  ; MOLD    CHANIGE OFF/ON  S/S
      RST     M670  ; Dummy   OK-Touch
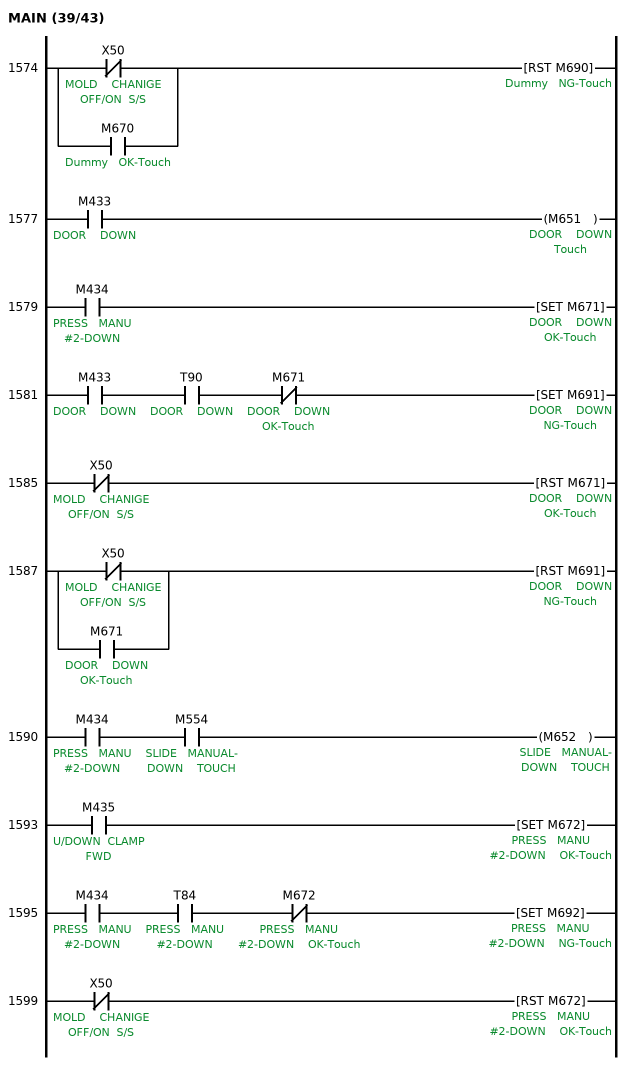
1574  LDI     X50  ; MOLD    CHANIGE OFF/ON  S/S
      OR      M670  ; Dummy   OK-Touch
      RST     M690  ; Dummy   NG-Touch
1577  LD      M433  ; DOOR    DOWN
      OUT     M651  ; DOOR    DOWN    Touch
1579  LD      M434  ; PRESS   MANU #2-DOWN
      SET     M671  ; DOOR    DOWN    OK-Touch
1581  LD      M433  ; DOOR    DOWN
      AND     T90  ; DOOR    DOWN
      ANI     M671  ; DOOR    DOWN    OK-Touch
      SET     M691  ; DOOR    DOWN    NG-Touch
1585  LDI     X50  ; MOLD    CHANIGE OFF/ON  S/S
      RST     M671  ; DOOR    DOWN    OK-Touch
1587  LDI     X50  ; MOLD    CHANIGE OFF/ON  S/S
      OR      M671  ; DOOR    DOWN    OK-Touch
      RST     M691  ; DOOR    DOWN    NG-Touch
1590  LD      M434  ; PRESS   MANU #2-DOWN
      AND     M554  ; SLIDE   MANUAL- DOWN    TOUCH
      OUT     M652  ; SLIDE   MANUAL- DOWN    TOUCH
1593  LD      M435  ; U/DOWN  CLAMP   FWD
      SET     M672  ; PRESS   MANU #2-DOWN    OK-Touch
1595  LD      M434  ; PRESS   MANU #2-DOWN
      AND     T84  ; PRESS   MANU #2-DOWN
      ANI     M672  ; PRESS   MANU #2-DOWN    OK-Touch
      SET     M692  ; PRESS   MANU #2-DOWN    NG-Touch
1599  LDI     X50  ; MOLD    CHANIGE OFF/ON  S/S
      RST     M672  ; PRESS   MANU #2-DOWN    OK-Touch
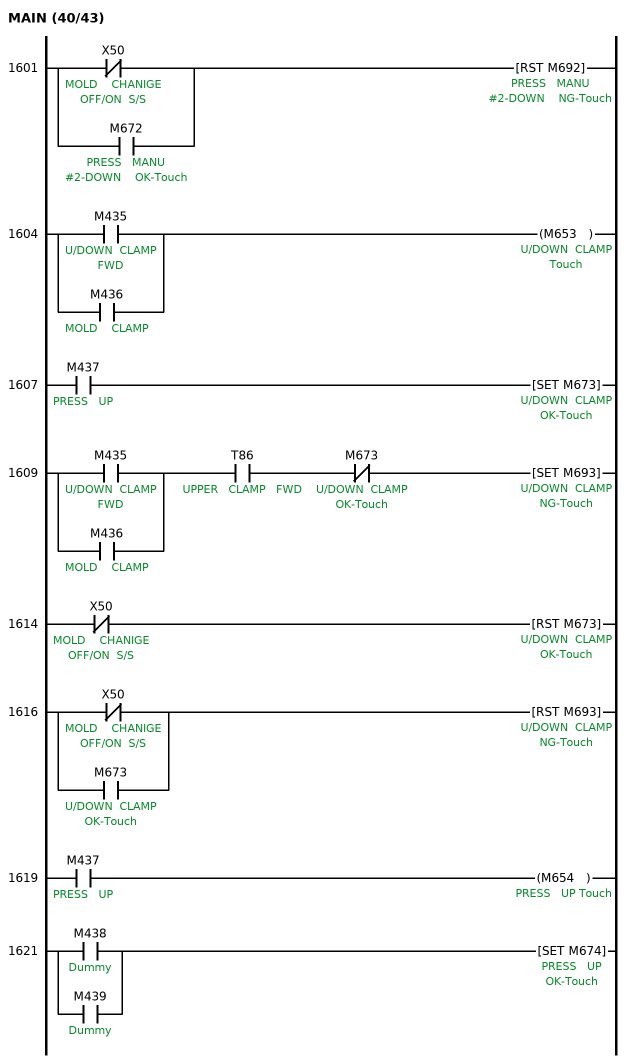
1601  LDI     X50  ; MOLD    CHANIGE OFF/ON  S/S
      OR      M672  ; PRESS   MANU #2-DOWN    OK-Touch
      RST     M692  ; PRESS   MANU #2-DOWN    NG-Touch
1604  LD      M435  ; U/DOWN  CLAMP   FWD
      OR      M436  ; MOLD    CLAMP
      OUT     M653  ; U/DOWN  CLAMP   Touch
1607  LD      M437  ; PRESS   UP
      SET     M673  ; U/DOWN  CLAMP   OK-Touch
1609  LD      M435  ; U/DOWN  CLAMP   FWD
      OR      M436  ; MOLD    CLAMP
      AND     T86  ; UPPER   CLAMP   FWD
      ANI     M673  ; U/DOWN  CLAMP   OK-Touch
      SET     M693  ; U/DOWN  CLAMP   NG-Touch
1614  LDI     X50  ; MOLD    CHANIGE OFF/ON  S/S
      RST     M673  ; U/DOWN  CLAMP   OK-Touch
1616  LDI     X50  ; MOLD    CHANIGE OFF/ON  S/S
      OR      M673  ; U/DOWN  CLAMP   OK-Touch
      RST     M693  ; U/DOWN  CLAMP   NG-Touch
1619  LD      M437  ; PRESS   UP
      OUT     M654  ; PRESS   UP Touch
1621  LD      M438  ; Dummy
      OR      M439  ; Dummy
      SET     M674  ; PRESS   UP      OK-Touch
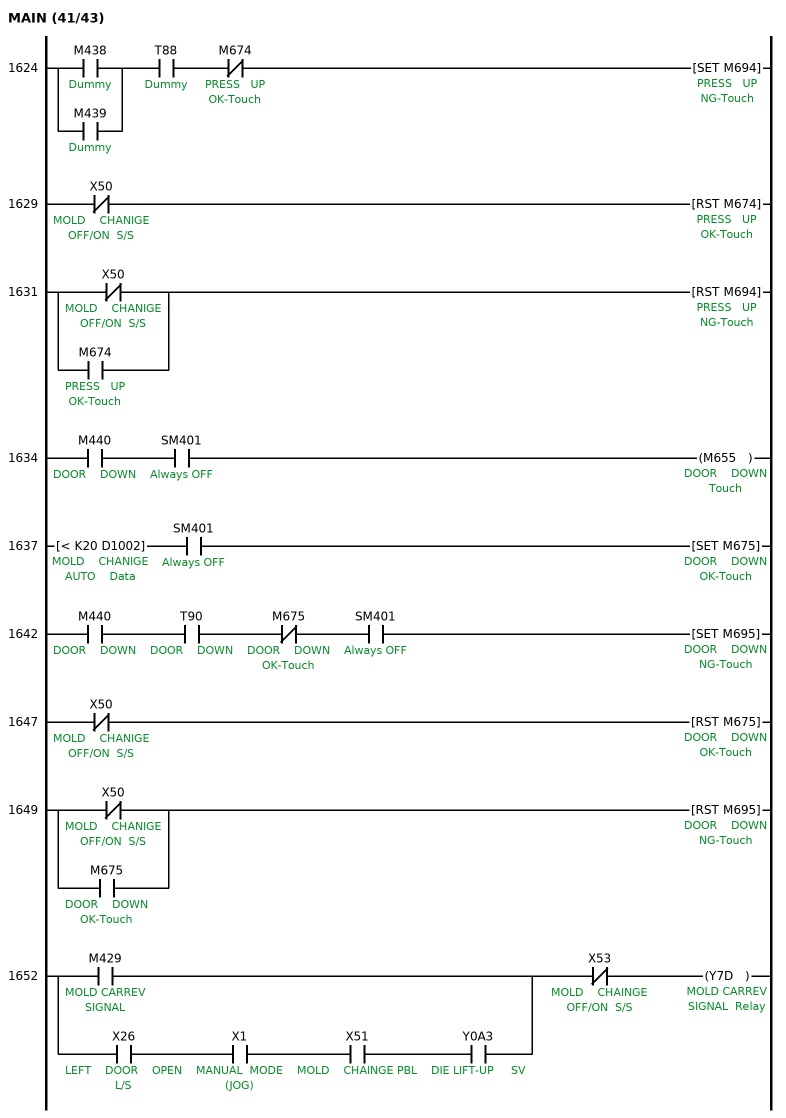
1624  LD      M438  ; Dummy
      OR      M439  ; Dummy
      AND     T88  ; Dummy
      ANI     M674  ; PRESS   UP      OK-Touch
      SET     M694  ; PRESS   UP      NG-Touch
1629  LDI     X50  ; MOLD    CHANIGE OFF/ON  S/S
      RST     M674  ; PRESS   UP      OK-Touch
1631  LDI     X50  ; MOLD    CHANIGE OFF/ON  S/S
      OR      M674  ; PRESS   UP      OK-Touch
      RST     M694  ; PRESS   UP      NG-Touch
1634  LD      M440  ; DOOR    DOWN
      AND     SM401  ; Always OFF
      OUT     M655  ; DOOR    DOWN    Touch
1637  LD<     K20 D1002  ; MOLD    CHANIGE AUTO    Data
      AND     SM401  ; Always OFF
      SET     M675  ; DOOR    DOWN    OK-Touch
1642  LD      M440  ; DOOR    DOWN
      AND     T90  ; DOOR    DOWN
      ANI     M675  ; DOOR    DOWN    OK-Touch
      AND     SM401  ; Always OFF
      SET     M695  ; DOOR    DOWN    NG-Touch
1647  LDI     X50  ; MOLD    CHANIGE OFF/ON  S/S
      RST     M675  ; DOOR    DOWN    OK-Touch
1649  LDI     X50  ; MOLD    CHANIGE OFF/ON  S/S
      OR      M675  ; DOOR    DOWN    OK-Touch
      RST     M695  ; DOOR    DOWN    NG-Touch
1652  LD      M429  ; MOLD CARREV     SIGNAL
      LD      X26  ; LEFT    DOOR    OPEN L/S
      AND     X1  ; MANUAL  MODE    (JOG)
      AND     X51  ; MOLD    CHAINGE PBL
      AND     Y0A3  ; DIE LIFT-UP     SV
      ORB
      ANI     X53  ; MOLD    CHAINGE OFF/ON  S/S
      OUT     Y7D  ; MOLD CARREV     SIGNAL  Relay
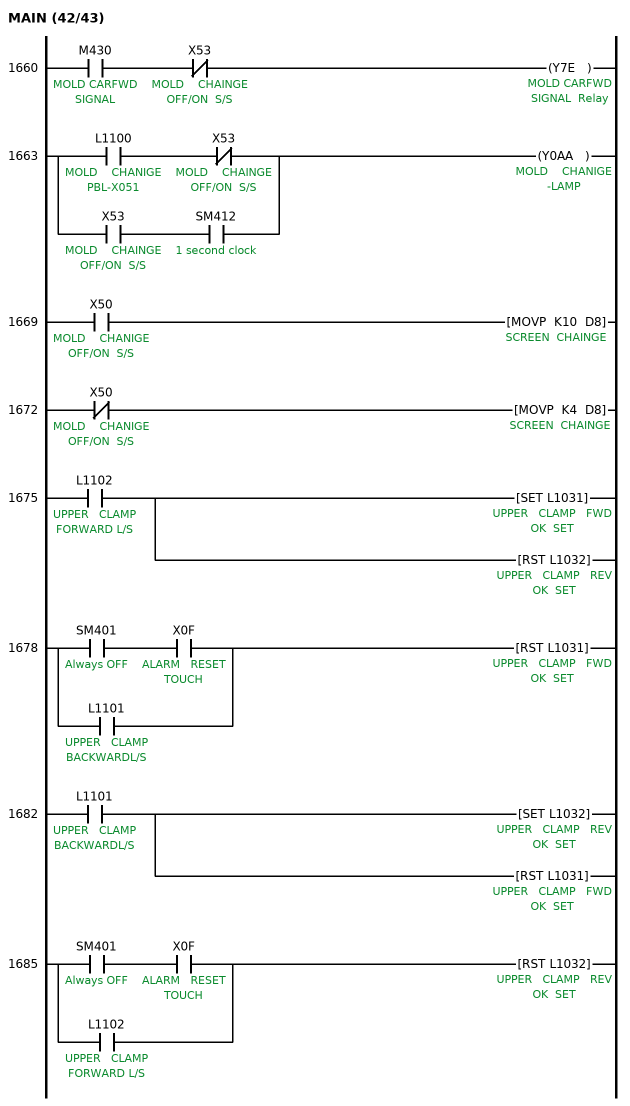
1660  LD      M430  ; MOLD CARFWD     SIGNAL
      ANI     X53  ; MOLD    CHAINGE OFF/ON  S/S
      OUT     Y7E  ; MOLD CARFWD     SIGNAL  Relay
1663  LD      L1100  ; MOLD    CHANIGE PBL-X051
      ANI     X53  ; MOLD    CHAINGE OFF/ON  S/S
      LD      X53  ; MOLD    CHAINGE OFF/ON  S/S
      AND     SM412  ; 1 second clock
      ORB
      OUT     Y0AA  ; MOLD    CHANIGE -LAMP
1669  LD      X50  ; MOLD    CHANIGE OFF/ON  S/S
      MOVP    K10 D8  ; SCREEN  CHAINGE
1672  LDI     X50  ; MOLD    CHANIGE OFF/ON  S/S
      MOVP    K4 D8
1675  LD      L1102  ; UPPER   CLAMP   FORWARD L/S
      SET     L1031  ; UPPER   CLAMP   FWD OK  SET
      RST     L1032  ; UPPER   CLAMP   REV OK  SET
1678  LD      SM401  ; Always OFF
      AND     X0F  ; ALARM   RESET   TOUCH
      OR      L1101  ; UPPER   CLAMP   BACKWARDL/S
      RST     L1031  ; UPPER   CLAMP   FWD OK  SET
1682  LD      L1101  ; UPPER   CLAMP   BACKWARDL/S
      SET     L1032  ; UPPER   CLAMP   REV OK  SET
      RST     L1031  ; UPPER   CLAMP   FWD OK  SET
1685  LD      SM401  ; Always OFF
      AND     X0F  ; ALARM   RESET   TOUCH
      OR      L1102  ; UPPER   CLAMP   FORWARD L/S
      RST     L1032  ; UPPER   CLAMP   REV OK  SET
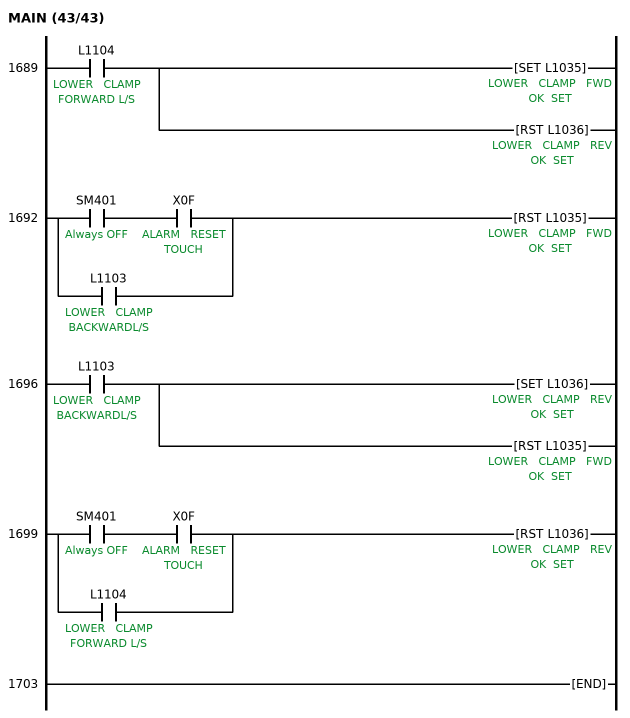
1689  LD      L1104  ; LOWER   CLAMP   FORWARD L/S
      SET     L1035  ; LOWER   CLAMP   FWD OK  SET
      RST     L1036  ; LOWER   CLAMP   REV OK  SET
1692  LD      SM401  ; Always OFF
      AND     X0F  ; ALARM   RESET   TOUCH
      OR      L1103  ; LOWER   CLAMP   BACKWARDL/S
      RST     L1035  ; LOWER   CLAMP   FWD OK  SET
1696  LD      L1103  ; LOWER   CLAMP   BACKWARDL/S
      SET     L1036  ; LOWER   CLAMP   REV OK  SET
      RST     L1035  ; LOWER   CLAMP   FWD OK  SET
1699  LD      SM401  ; Always OFF
      AND     X0F  ; ALARM   RESET   TOUCH
      OR      L1104  ; LOWER   CLAMP   FORWARD L/S
      RST     L1036  ; LOWER   CLAMP   REV OK  SET
1703  END
END_PROGRAM

// device comments not shown above
X3  ; STOP MODE
X6  ; PANEL   START   TOUCH
X31  ; START B FROM ROBOT
X39  ; LOWER CLAMP PRESSURE SWITCH
X3A  ; DIE LIFT PRESSURE SWITCH
Y0A8  ; Y7D
